INTERFACE ITF_2_6AxisRobot EXTENDS ITF_1_Robot

METHOD Home : BOOL
VAR_INPUT
END_VAR
END_METHOD

METHOD MoveJoint : BOOL
VAR_INPUT
    joints : stJoint6;
END_VAR
END_METHOD

METHOD MoveJointRelative : BOOL
VAR_INPUT
    offsets : stJoint6;
END_VAR
END_METHOD

METHOD MoveLinear : BOOL
VAR_INPUT
    target : stTarget3D;
END_VAR
END_METHOD

METHOD MoveLinearRelative : BOOL
  VAR_INPUT
    offset : stRelativePose3D;
  END_VAR
END_METHOD

METHOD SetTool : BOOL
VAR_INPUT
    tool : FB_Tool;
END_VAR
END_METHOD

METHOD SetFrame : BOOL
VAR_INPUT
    frame : stFrame;
END_VAR
END_METHOD

{warning 'Eigenschaftenimplementierung hinzufügen'}
PROPERTY ActualJointPosition : stJoint6
GET
END_GET
END_PROPERTY

PROPERTY ActualJointVelocity : stJoint6
GET
END_GET
END_PROPERTY

{warning 'Eigenschaftenimplementierung hinzufügen'}
PROPERTY ActualTcpPose : stPose3D
GET
END_GET
END_PROPERTY

PROPERTY ActualTcpVelocity : stPose3D
GET
END_GET
END_PROPERTY

PROPERTY CurrentFrame : stFrame
GET
END_GET
SET
END_SET
END_PROPERTY

PROPERTY CurrentFrameId : UINT
GET
END_GET
END_PROPERTY

PROPERTY CurrentTool : FB_Tool
GET
END_GET
SET
END_SET
END_PROPERTY

PROPERTY IsHomePosition : BOOL
GET
END_GET
END_PROPERTY

{warning 'Add property implementation'}
PROPERTY TargetReached : BOOL
GET
END_GET
END_PROPERTY

END_INTERFACE

(* stored: Version 1.1.0.1, ProductVersion 3.1.4026.18
   Itf ITF_2_6AxisRobot: Id {5597e200-2768-442d-a894-79ed17b4bd75}
   Method Home: Id {9008c31c-e8e7-4fc4-ab50-fce636f66aa9}
   Method MoveJoint: Id {01831dea-3b4d-496c-9028-1a30987f2ab5}
   Method MoveJointRelative: Id {0f521464-ec50-448d-bb07-d37ea83816d3}
   Method MoveLinear: Id {617f15d3-641e-4bd1-b8bf-7e1c16712ddc}
   Method MoveLinearRelative: Id {bdfb6932-6a17-4ad8-a206-492214d6a04f}
   Method SetTool: Id {4419060a-b81d-49ba-98b5-0e9531683def}
   Method SetFrame: Id {4f810bbe-4c7e-4ed8-a1f1-65b416f3d016}
   Property ActualJointPosition: Id {f4e9d5a1-845e-4b46-b1f5-b6013f3c1bf2}
   Get Get: Id {9bc35bbe-7807-471e-9049-dfe1eaeec2ec}
   Property ActualJointVelocity: Id {a5ea3d6b-243a-4425-9bdd-13270e6b23d8}
   Get Get: Id {b2cbd5f6-df64-4021-8c9b-d68ee343f3fa}
   Property ActualTcpPose: Id {3ccb050e-fb6b-4d88-80e5-9740c700b585}
   Get Get: Id {26f7e51c-a2e1-4966-939c-6ce06ce2cce5}
   Property ActualTcpVelocity: Id {29c2cbff-861a-434c-bd80-cca88e4b0432}
   Get Get: Id {d62f14c4-b447-4702-98b3-1685b412e392}
   Property CurrentFrame: Id {37fb2f8c-1107-4f5c-8321-fe9b2b8c3eac}
   Get Get: Id {483c18a1-b1a6-4612-8bab-6f52b909a18d}
   Set Set: Id {93b7ec30-7f1c-471f-9a92-dce39896542d}
   Property CurrentFrameId: Id {b512308c-5850-48a7-85d0-fd48d82becb3}
   Get Get: Id {e164a528-6e1a-43c4-9de7-0c89ea47d23b}
   Property CurrentTool: Id {31260ea4-d74c-4661-b977-2f4fbc51c3ad}
   Get Get: Id {50378180-4e1c-40ab-b830-dd6d8d1d884b}
   Set Set: Id {66ad7fee-1b3e-4673-8360-95856cb39db8}
   Property IsHomePosition: Id {70f6bdc3-81d8-4a72-9961-a731a8f684fb}
   Get Get: Id {376ed0f7-d8a4-4e9c-ac1b-17426e13c0b7}
   Property TargetReached: Id {5f879bbf-7361-48f8-9f67-1ba39a94979d}
   Get Get: Id {2a36317c-e606-43b2-a57c-1527af6e3f25} *)
